// TIA Portal V18 export
FUNCTION_BLOCK "ZAxis_RelativeMotion_Test"   // FB25, LAD
{ S7_Optimized_Access := 'TRUE' }
VERSION : 0.1
// stored: AutoNumber true, IsIECCheckEnabled false, IsRetainMemResEnabled false, MemoryReserve 100, SetENOAutomatically false, UDAEnableTagReadback false
   VAR_INPUT
      StartTest : Bool;
      EndTest : Bool;
      AmountOfSteps : DInt := 3000;
      StepSizeInput : DInt := 100;
      Position : DInt := 0;
      AxisMoving : Bool;
   END_VAR
   VAR_OUTPUT
      StartTask : Bool;
      StepSize : DInt;
      StepNumber : DInt;
      CreateLogFile : Bool;
      StartLog : Bool;
      Comment : String;
   END_VAR
   VAR
      TestActiveInternal : Bool;
      ActualStep : DInt := 9999;
      StepCountNext : DInt := 1;
      MovingInternal : Bool;
      ChangingCount : Bool;
      StartTaskM : Bool;
      LogCreatingReady : Bool;
   END_VAR
BEGIN

REGION Network 1: Log Creating
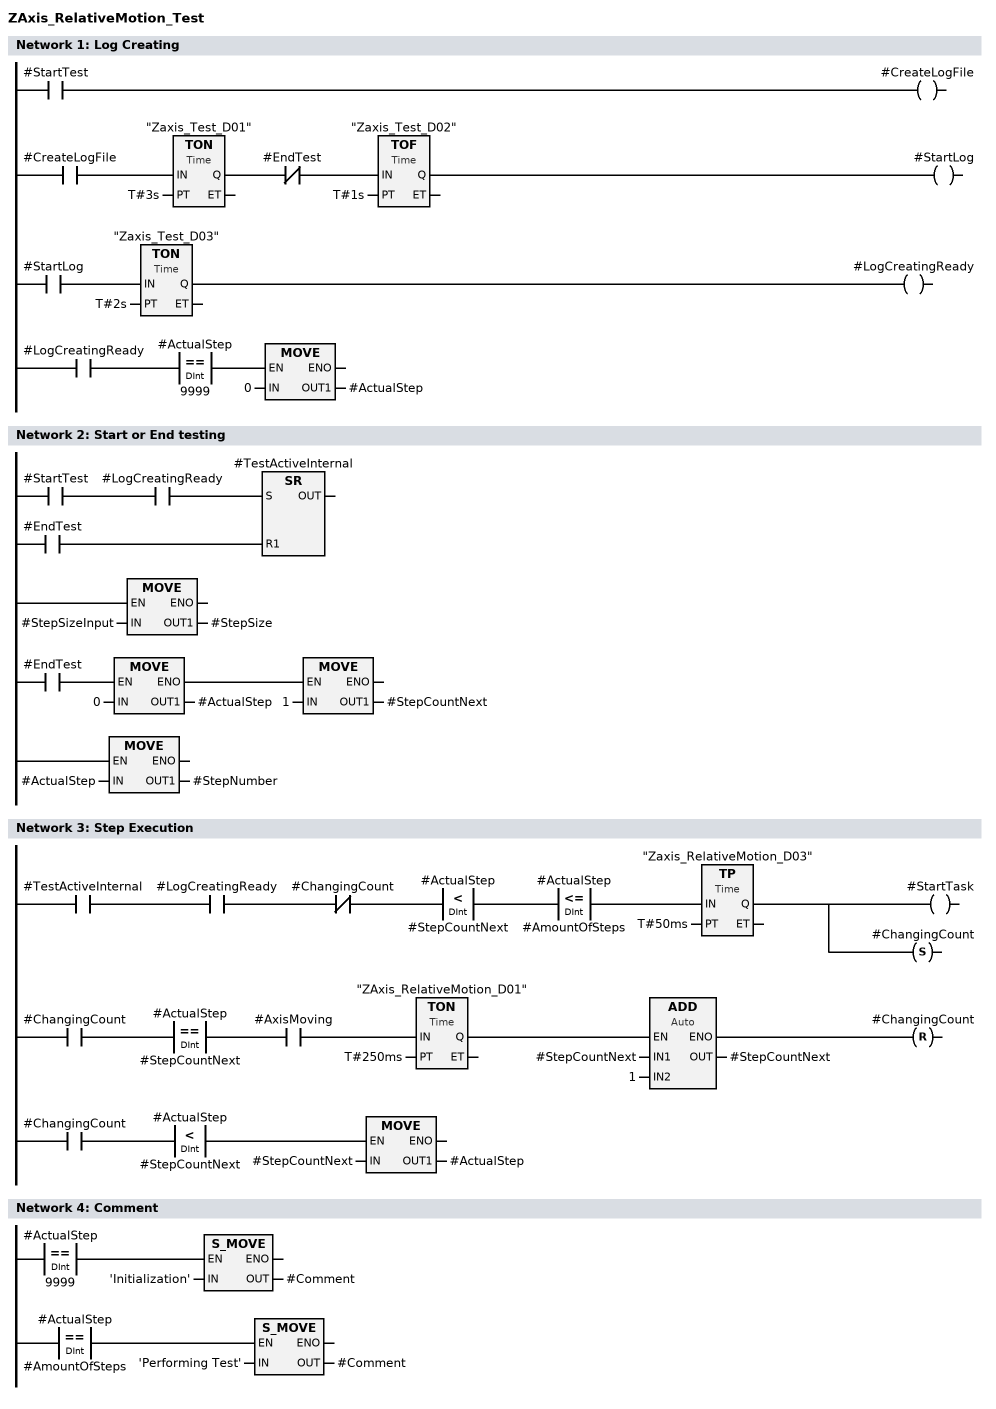
   RUNG wire#powerrail
      Contact( #StartTest )
      Coil( #CreateLogFile )
   END_RUNG
   RUNG wire#powerrail
      Contact( #CreateLogFile )
      { S7_Templates := "time_type := Time" } "Zaxis_Test_D01".TON(pt := T#3s, et =>)
      I_Contact( #EndTest )
      { S7_Templates := "time_type := Time" } "Zaxis_Test_D02".TOF(pt := T#1s, et =>)
      Coil( #StartLog )
   END_RUNG
   RUNG wire#powerrail
      Contact( #StartLog )
      { S7_Templates := "time_type := Time" } "Zaxis_Test_D03".TON(pt := T#2s, et =>)
      Coil( #LogCreatingReady )
   END_RUNG
   RUNG wire#powerrail
      Contact( #LogCreatingReady )
      { S7_Templates := "SrcType := DInt" } EQ_Contact(in1 := #ActualStep, in2 := 9999)
      Move(in := 0, out1 => #ActualStep)
   END_RUNG
   // the same network as SCL:
   #CreateLogFile := #StartTest;
   "Zaxis_Test_D01".TON(IN := #CreateLogFile, PT := T#3s);
   "Zaxis_Test_D02".TOF(IN := "Zaxis_Test_D01".Q AND NOT #EndTest, PT := T#1s);
   #StartLog := "Zaxis_Test_D02".Q;
   "Zaxis_Test_D03".TON(IN := #StartLog, PT := T#2s);
   #LogCreatingReady := "Zaxis_Test_D03".Q;
   IF #LogCreatingReady AND (#ActualStep = 9999) THEN #ActualStep := 0; END_IF;
END_REGION

REGION Network 2: Start or End testing
   RUNG wire#powerrail
      Contact( #StartTest )
      Contact( #LogCreatingReady )
      S_SR(operand := #TestActiveInternal, r1 := wire#w1)
   END_RUNG
   RUNG wire#powerrail
      Contact( #EndTest )
   END_RUNG wire#w1
   RUNG wire#powerrail
      Move(in := #StepSizeInput, out1 => #StepSize)
   END_RUNG
   RUNG wire#powerrail
      Contact( #EndTest )
      Move(in := 0, out1 => #ActualStep)
      Move(in := 1, out1 => #StepCountNext)
   END_RUNG
   RUNG wire#powerrail
      Move(in := #ActualStep, out1 => #StepNumber)
   END_RUNG
   // the same network as SCL:
   IF #StartTest AND #LogCreatingReady THEN
       #TestActiveInternal := TRUE;   // SR flip-flop
   END_IF;
   IF #EndTest THEN #TestActiveInternal := FALSE; END_IF;
   #StepSize := #StepSizeInput;
   IF #EndTest THEN
       #ActualStep := 0;
       #StepCountNext := 1;
   END_IF;
   #StepNumber := #ActualStep;
END_REGION

REGION Network 3: Step Execution
   RUNG wire#powerrail
      Contact( #TestActiveInternal )
      Contact( #LogCreatingReady )
      I_Contact( #ChangingCount )
      { S7_Templates := "SrcType := DInt" } LT_Contact(in1 := #ActualStep, in2 := #StepCountNext)
      { S7_Templates := "SrcType := DInt" } LE_Contact(in1 := #ActualStep, in2 := #AmountOfSteps)
      { S7_Templates := "time_type := Time" } "Zaxis_RelativeMotion_D03".TP(pt := T#50ms, et =>)
      wire#w1
      Coil( #StartTask )
   END_RUNG
   RUNG wire#w1
      S_Coil( #ChangingCount )
   END_RUNG
   RUNG wire#powerrail
      Contact( #ChangingCount )
      { S7_Templates := "SrcType := DInt" } EQ_Contact(in1 := #ActualStep, in2 := #StepCountNext)
      Contact( #AxisMoving )
      { S7_Templates := "time_type := Time" } "ZAxis_RelativeMotion_D01".TON(pt := T#250ms, et =>)
      Add(in1 := #StepCountNext, in2 := 1, out => #StepCountNext)
      R_Coil( #ChangingCount )
   END_RUNG
   RUNG wire#powerrail
      Contact( #ChangingCount )
      { S7_Templates := "SrcType := DInt" } LT_Contact(in1 := #ActualStep, in2 := #StepCountNext)
      Move(in := #StepCountNext, out1 => #ActualStep)
   END_RUNG
   // the same network as SCL:
   "Zaxis_RelativeMotion_D03".TP(IN := #TestActiveInternal AND #LogCreatingReady AND NOT #ChangingCount AND (#ActualStep < #StepCountNext) AND (#ActualStep <= #AmountOfSteps),
                           PT := T#50ms);
   #StartTask := "Zaxis_RelativeMotion_D03".Q;
   IF "Zaxis_RelativeMotion_D03".Q THEN #ChangingCount := TRUE; END_IF;
   "ZAxis_RelativeMotion_D01".TON(IN := #ChangingCount AND (#ActualStep = #StepCountNext) AND #AxisMoving,
                           PT := T#250ms);
   IF "ZAxis_RelativeMotion_D01".Q THEN
       #StepCountNext := #StepCountNext + 1;
       #ChangingCount := FALSE;
   END_IF;
   IF #ChangingCount AND (#ActualStep < #StepCountNext) THEN #ActualStep := #StepCountNext; END_IF;
END_REGION

REGION Network 4: Comment
   RUNG wire#powerrail
      { S7_Templates := "SrcType := DInt" } EQ_Contact(in1 := #ActualStep, in2 := 9999)
      S_Move(in := 'Initialization', out => #Comment)
   END_RUNG
   RUNG wire#powerrail
      { S7_Templates := "SrcType := DInt" } EQ_Contact(in1 := #ActualStep, in2 := #AmountOfSteps)
      S_Move(in := 'Performing Test', out => #Comment)
   END_RUNG
   // the same network as SCL:
   IF #ActualStep = 9999 THEN #Comment := 'Initialization'; END_IF;
   IF #ActualStep = #AmountOfSteps THEN #Comment := 'Performing Test'; END_IF;
END_REGION
END_FUNCTION_BLOCK
